{attribute 'qualified_only'}
{attribute 'strict'}
TYPE E_Joystick :
(
	enum_member := 0
);
END_TYPE

(* stored: Version 1.1.0.1, ProductVersion 3.1.4024.10
   DUT E_Joystick: Id {9a4fcfb2-fd86-492c-9edd-f8bb75a4e83a} *)
